{attribute 'linkalways'} 
{attribute 'no_explicit_call' := 'This FB is a CLASS and must be accessed using methods or properties'}
{attribute 'enable_dynamic_creation'}
FUNCTION_BLOCK _TcVnVector2_USINT EXTENDS AliasDatatypeBase
VAR
	localData : TcVnVector2_USINT;
	activeData : REFERENCE TO TcVnVector2_USINT REF= localData;
	aliasBaseDatatype : _Array0to1OfUSINT;
END_VAR

PROPERTY PUBLIC Address : PVOID
GET
Address := ADR(activeData);
END_GET
END_PROPERTY

METHOD PUBLIC ClearReference
VAR_INPUT
END_VAR
activeData REF= localData;
SetBaseDatatypeReference();
END_METHOD

METHOD PUBLIC Clone : I_Datatype
VAR
    pClone : POINTER TO _TcVnVector2_USINT;
END_VAR
pClone := __NEW(_TcVnVector2_USINT);
Clone := pClone^;
END_METHOD

METHOD FB_init : BOOL
VAR_INPUT
	bInitRetains : BOOL; // if TRUE, the retain variables are initialized (warm start / cold start)
	bInCopyCode : BOOL;  // if TRUE, the instance afterwards gets moved into the copy code (online change)
	//InitialValue : <type>; // if possible, not all values can be initialized
END_VAR
//localData := InitialValue; // if possible, not all values can be initialized
SetBaseDatatypeReference();
AddBaseDatatype(aliasBaseDatatype);
END_METHOD

PROPERTY PUBLIC Identifier : T_MAXSTRING
GET
Identifier := 'TcVnVector2_USINT';
END_GET
END_PROPERTY

METHOD PUBLIC MakeReferenceTo
VAR_INPUT
	ReferenceTarget : REFERENCE TO TcVnVector2_USINT;
END_VAR
activeData REF= ReferenceTarget;
SetBaseDatatypeReference();
END_METHOD

METHOD PROTECTED SetBaseDatatypeReference
VAR_INPUT
END_VAR
aliasBaseDatatype.MakeReferenceTo(activeData);
END_METHOD

PROPERTY PUBLIC Size : UDINT
GET
Size := SIZEOF(activeData);
END_GET
END_PROPERTY

METHOD TryMakeReferenceTo : BOOL
VAR_INPUT
	Target : I_Datatype;
END_VAR
VAR
	pTargetData : POINTER TO TcVnVector2_USINT;
END_VAR
IF NOT IsEquivalentTo(Target) THEN
	RETURN;
END_IF

pTargetData := Target.Address;
activeData REF= pTargetData^;
SetBaseDatatypeReference();
TryMakeReferenceTo := TRUE;
END_METHOD

PROPERTY PUBLIC Value : REFERENCE TO TcVnVector2_USINT
GET
Value REF= activeData;
END_GET
END_PROPERTY

END_FUNCTION_BLOCK

(* stored: Version 1.1.0.1, ProductVersion 3.1.4024.13
   POU _TcVnVector2_USINT: Id {ada535f2-5aeb-0918-066d-69d2c2ac3135}, SpecialFunc None
   Folder Core: Id {bf434c4d-4916-03fa-20fe-30378f6f9386}
   Folder Protected: Id {9f0b1118-038f-0ce8-3637-5aecb7513676}
   Folder Customize: Id {8291e76a-f484-0e0b-143b-811ea509cc21}
   Folder Constructor: Id {cf3f9585-640e-0ee8-1737-2c27429cce92}
   Property Address: Id {4a65ac9d-1407-0912-0e79-e67956729817}
   Get Get: Id {41b5389c-7409-0f0f-1872-aa80973d8daa}
   Method ClearReference: Id {76b084ef-d8cc-057d-25ec-b591cc72c417}
   Method Clone: Id {b49996b5-2309-047d-1a39-21bae1b2e2e6}
   Method FB_init: Id {e6d12f28-2437-0173-2b5b-5fc67ff59a20}
   Property Identifier: Id {02d76903-a60f-02b6-3c32-baf6ad8cb7e9}
   Get Get: Id {ba2ada73-a2f5-0c73-32a1-265f82972279}
   Method MakeReferenceTo: Id {52239def-dc5e-0bdb-2db5-c101a57bf8a4}
   Method SetBaseDatatypeReference: Id {a0e0c1bb-6c00-0a2c-0447-5c2e8dbf525b}
   Property Size: Id {40cd4906-18fb-03c7-2ed6-3c1659fb2252}
   Get Get: Id {cac087c7-c43e-0593-0a4b-3bb9042a745e}
   Method TryMakeReferenceTo: Id {4349d706-fab2-06ab-3a13-d7a4d7220e0f}
   Property Value: Id {91e43ae6-65e9-0f97-0c31-41fffdf29865}
   Get Get: Id {5578d49a-d9f3-0e90-1fa7-911e8bebcc27} *)
